// TIA Portal V20 export
DATA_BLOCK "IDB_PackedLine"   // DB10
// stored: Access Published, InstanceOfName PackedLine.FB_PackedLine, InstanceOfType FB, Namespace PackedLine
"PackedLine.FB_PackedLine"
   // VAR
   //    "G1.1.1" { S7_SetPoint := 'True'} : "Global.FB_Conveyor";
   //    "G1.1.2" { S7_SetPoint := 'True'} : "Global.FB_Conveyor";
   //    "G1.1.3" { S7_SetPoint := 'True'} : "Global.FB_Conveyor";
   //    "G1.1.4" { S7_SetPoint := 'True'} : "Global.FB_Conveyor";
   //    "G1.1.5" { S7_SetPoint := 'True'} : "Global.FB_Conveyor";
   //    "G1.1.6" { S7_SetPoint := 'True'} : "Global.FB_Conveyor";
   //    "G1.1.7" { S7_SetPoint := 'True'} : "Global.FB_Conveyor";
   //    "G1.1.8" { S7_SetPoint := 'True'} : "Global.FB_Conveyor";
   //    "G1.1.9" { S7_SetPoint := 'True'} : "Global.FB_Conveyor";
   //    "G1.1.10" { S7_SetPoint := 'True'} : "Global.FB_Conveyor";
   //    "G1.1.11" { S7_SetPoint := 'True'} : "Global.FB_Conveyor";
   //    "G1.1.12" { S7_SetPoint := 'True'} : "Global.FB_Conveyor";
   //    "G1.1.13" { S7_SetPoint := 'True'} : "Global.FB_Conveyor";
   //    "G1.1.14" { S7_SetPoint := 'True'} : "Global.FB_Conveyor";
   //    "G1.1.15" { S7_SetPoint := 'True'} : "Global.FB_Conveyor";
   //    "G1.1.16" { S7_SetPoint := 'True'} : "Global.FB_Conveyor";
   //    "G1.1.17" { S7_SetPoint := 'True'} : "Global.FB_Conveyor";
   //    "G1.1.18" { S7_SetPoint := 'True'} : "Global.FB_Conveyor";
   //    "G1.1.19" { S7_SetPoint := 'True'} : "Global.FB_Conveyor";
   //    "G1.2.1" { S7_SetPoint := 'True'} : "Global.FB_Conveyor";
   //    "G1.2.2" { S7_SetPoint := 'True'} : "Global.FB_Conveyor";
   //    "G1.3.1" { S7_SetPoint := 'True'} : "Global.FB_Conveyor";
   //    "G1.4.1" { S7_SetPoint := 'True'} : "Global.FB_Conveyor";
   //    "G1.4.2" { S7_SetPoint := 'True'} : "Global.FB_Conveyor";
   //    "G1.4.3" { S7_SetPoint := 'True'} : "Global.FB_Conveyor";
   //    "G1.4.4" { S7_SetPoint := 'True'} : "Global.FB_Conveyor";
   //    "G1.4.5" { S7_SetPoint := 'True'} : "Global.FB_Conveyor";
   //    "G1.4.6" { S7_SetPoint := 'True'} : "Global.FB_Conveyor";
   //    "G1.5.1" { S7_SetPoint := 'True'} : "Global.FB_Conveyor";
   //    "G1.5.2" { S7_SetPoint := 'True'} : "Global.FB_Conveyor";
   //    "G1.5.3" { S7_SetPoint := 'True'} : "Global.FB_Conveyor";
   //    "G1.5.4" { S7_SetPoint := 'True'} : "Global.FB_Conveyor";
   //    "G1.5.5" { S7_SetPoint := 'True'} : "Global.FB_Conveyor";
   //    "G1.5.6" { S7_SetPoint := 'True'} : "Global.FB_Conveyor";
   //    "G1.6.1" { S7_SetPoint := 'True'} : "Global.FB_Conveyor";
   //    "G1.6.2" { S7_SetPoint := 'True'} : "Global.FB_Conveyor";
   //    "G1.7.1" { S7_SetPoint := 'True'} : "Global.FB_Conveyor";
   //    "G1.7.2" { S7_SetPoint := 'True'} : "Global.FB_Conveyor";
   //    "G1.7.3" { S7_SetPoint := 'True'} : "Global.FB_Conveyor";
   //    "G1.7.4" { S7_SetPoint := 'True'} : "Global.FB_Conveyor";
   // END_VAR
BEGIN
END_DATA_BLOCK
